PROGRAM MAIN
VAR

END_VAR

// ***********************************************************************************
//
// Müller-steinag Gruppe, Kandergrien Einigen, CH-3646 Bern
// ETH Zurich, Building HIF E26, Laura-Hezner-Weg 7, CH-8093 Zürich
// 
// ***********************************************************************************
// 
// PROJECT     :  A061 Digital Casting System 
// FUNCTION    :  Main 
// AUTHOR      :  Weiting Chen
// EMAIL       :  chenw@usi.ch
// Copyright   :  USI Mendrisio; ETH Zürich; Müller-steinag Gruppe (CH) 2024
//
// ***********************************************************************************


P_Control_Mode();

// data comunicaiton robot via EL6631

IF GVL.b_mode_laptop THEN 
	P_Laptop_Operate();
ELSIF GVL.b_mode_robot THEN 
	P_PNDataConvert();
	P_Robot_Operate();
ELSIF GVL.b_mode_manual THEN 
	P_Manual_Operate();
END_IF


// ELSE
// 	temp_speed_override:=F_ScalAnalogOut(
// 		n_Input:= REAL_TO_INT(GVL_IO.in_MI1_Poti_Speed),
// 		n_InMin:= 0,
// 		n_InMax:= 32767,
// 		n_OutMin:= 0,
// 		n_OutMax:= 100);
// END_IF

// GVL_VAR.f_MI1_Override:= temp_speed_override;

END_PROGRAM

(* stored: Version 1.2.0.0, ProductVersion 3.1.4024.11
   POU MAIN: Id {aa6047d7-dda4-4a4e-8872-4170f9749e6f}, SpecialFunc None *)
